(* IEC 61131-3 sources: mastertool-rankine-bridge/tests/indexer/fixtures/sample_export/objects/application_prg_1__PrgResolucaoSintetica, 2 files *)

(* ---- declaration.st ---- *)
PROGRAM PrgResolucaoSintetica
VAR
    MT01            : BOOL;
    fbTimer         : FB_TimerSintetico;
    tTempoAjustado   : TIME;
    xPulso          : BOOL;
END_VAR

(* ---- implementation.st ---- *)
MT01 := TRUE;

GvlDiagnosticoSintetico.DG_Contador := 1;

IF GA_ValorSintetico > 0 THEN
    xPulso := TRUE;
END_IF;

IF DG_Contador > 0 THEN
    xPulso := TRUE;
END_IF;

fbTimer(
    xStart := xPulso,
    tPreset := tTempoAjustado,
    xDone => xPulso
);

fbTimer.Reset();
